FUNCTION_BLOCK Station EXTENDS CyclicBase IMPLEMENTS IStation
VAR_INPUT
END_VAR
VAR_OUTPUT
END_VAR
VAR
	_Empty : BOOL;
	_Complete : BOOL;
	_Operating : BOOL;
	_Ready : BOOL;
	_Positions : ARRAY[1..4] OF MC_LREAL := [0.0,0.0,0.0,0.0];
	NumberOfPositions : INT := 0;
	AssignedPositions : INT := 1;
	StationMovers : INT;
	stInfo : stStationInfo;
	_HasMover : BOOL;
	ProductCounter : R_TRIG;
	Products : DINT;
	LastStation : BOOL;
	MyMover : IMover;
END_VAR

{analysis -2}

METHOD Abort : BOOL
VAR_INPUT
END_VAR
_Complete := FALSE;
_Empty := TRUE;
_Operating := FALSE;
_Ready := TRUE;
Abort := true;
END_METHOD

METHOD PUBLIC  Cycle : HRESULT
VAR_INPUT
END_VAR
//Cyclic info
stInfo.StationPosition := _Positions[1];
stInfo.StationStatus.Empty := _Empty;
stInfo.StationStatus.Complete := _Complete;
stInfo.StationStatus.HasMover := _HasMover;
stInfo.StationStatus.Operating := _Operating;
stInfo.StationStatus.Ready := _Ready;

IF LastStation THEN
	ProductCounter(CLK := _Complete);
	IF ProductCounter.Q THEN
		Products := Products + 1;
	END_IF
END_IF

Cycle := S_OK;
END_METHOD

METHOD HasMover : BOOL
VAR_INPUT
	mover : IMover;
END_VAR
StationMovers := StationMovers + 1;
IF StationMovers = NumberOfPositions THEN
	_HasMover := TRUE;
END_IF
MyMover := mover;
HasMover := TRUE;
END_METHOD

METHOD IsClear : BOOL
IsClear := _Empty;
END_METHOD

METHOD isComplete : BOOL
isComplete := _Complete;
END_METHOD

PROPERTY PUBLIC IsLastStation : BOOL
GET
IsLastStation := LastStation;
END_GET
SET
LastStation := IsLastStation;
END_SET
END_PROPERTY

METHOD IsOperating : BOOL
IsOperating := _Operating;
END_METHOD

METHOD IsReady : BOOL
IsReady := _Ready;
END_METHOD

METHOD MoverAway : BOOL
VAR_INPUT
END_VAR
StationMovers := StationMovers - 1;
MyMover := 0;
MoverAway := TRUE;
END_METHOD

PROPERTY Position : MC_LREAL
GET
Position := _Positions[AssignedPositions];
AssignedPositions := AssignedPositions + 1;
IF AssignedPositions > NumberOfPositions THEN
	AssignedPositions := 1;
END_IF
END_GET
SET
IF NumberOfPositions < 5 THEN
	NumberOfPositions := NumberOfPositions + 1;
	_Positions[NumberOfPositions] := Position;
END_IF
END_SET
END_PROPERTY

END_FUNCTION_BLOCK

(* stored: Version 1.1.0.1, ProductVersion 3.1.4024.12
   POU Station: Id {506a1b5f-d283-4b99-9adf-318a9c36fdac}, SpecialFunc None
   Method Abort: Id {b49ff0e5-eb8b-49bd-befd-0bab45ac01fe}
   Method Cycle: Id {718bc2ed-83e9-4df0-b688-ff0112cf7157}
   Method HasMover: Id {cfa7f397-450b-4982-8373-384ee5df1767}
   Method IsClear: Id {5a1d616a-dcb0-4a56-9caf-0526ba7a4fac}
   Method isComplete: Id {5a7054f2-4dbb-4c61-9bd3-b1648c0eccb5}
   Property IsLastStation: Id {bd96d050-990a-4fff-89e6-b506df6988f2}
   Get Get: Id {6a265c68-4fa4-453c-a40c-d846a57c2b37}
   Set Set: Id {4793574b-7d23-4a86-a240-9dc35ed22c28}
   Method IsOperating: Id {5d80dcb3-b05c-443a-91b8-3bed25c3df07}
   Method IsReady: Id {030f67f6-2ceb-4b14-bbf0-d64116218e04}
   Method MoverAway: Id {6941b853-93be-47e5-be62-9ae205bb30c2}
   Property Position: Id {e826f73c-3eb0-49b1-8a82-785d3b45b5a4}
   Get Get: Id {28648367-e6e3-4e2f-bc66-080beef37026}
   Set Set: Id {c5e3a131-a10c-4d0d-ac13-bde814ce94ed} *)
